FUNCTION_BLOCK FB_Lift EXTENDS FB_BaseDevice

VAR
	fbServo: FB_SEW_MovidriveB;
END_VAR

VAR PERSISTENT
	bAbove_1_or_Below_0_HomePos: BOOL;
	bExtending_1_or_Retracting_0: BOOL;
	eSMState: (INIT, ENABLE, MOVE_TRIG, MOVING, MOVED, STOP, ERROR, RESET) := INIT;
	nGearRation: REAL; 
	nInertia: REAL;
END_VAR

END_FUNCTION_BLOCK

(* stored: Version 1.1.0.1, ProductVersion 3.1.4024.12
   POU FB_Lift: Id {20d4ee3a-b9db-4f8a-8627-ecd4d53597db}, SpecialFunc None *)
